TYPE csp_case_flap_control_connection_status_enum :
(		
	CSP_CASE_FLAP_CONTROL_STATUS_CONNECTION_START					:= 0,
	CSP_CASE_FLAP_CONTROL_STATUS_CONNECTION_ENGAGE					:= 10,
	CSP_CASE_FLAP_CONTROL_STATUS_CONNECTION_ENGAGED					:= 20,
	CSP_CASE_FLAP_CONTROL_STATUS_CONNECTION_CHECK_CHANGE_CAM			:= 30,
	CSP_CASE_FLAP_CONTROL_STATUS_CONNECTION_CHANGE_CAM				:= 40,
	CSP_CASE_FLAP_CONTROL_STATUS_CONNECTION_WAIT_NEW_CAM				:= 50,
	CSP_CASE_FLAP_CONTROL_STATUS_CONNECTION_DONE 					:= 900,
	CSP_CASE_FLAP_CONTROL_STATUS_CONNECTION_ERROR 					:= 999
) := CSP_CASE_FLAP_CONTROL_STATUS_CONNECTION_START;
END_TYPE

(* stored: Version 1.1.0.1, ProductVersion 3.1.4024.3
   DUT csp_case_flap_control_connection_status_enum: Id {6d743088-d4ec-062b-2d96-005f1cd75ca0} *)
